FUNCTION_BLOCK PusherControl (* Basic Function Block Type *)
  (* Standard: 61499-2 *)
  (* Version 0.0, 1/14/2024, midxav, Template *)
  PACKAGE Main;
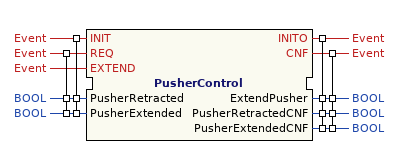
  EVENT_INPUT
    INIT WITH PusherRetracted, PusherExtended; (* Initialization Request *)
    REQ WITH PusherRetracted, PusherExtended; (* Normal Execution Request *)
    EXTEND;
  END_EVENT
  EVENT_OUTPUT
    INITO WITH ExtendPusher, PusherRetractedCNF, PusherExtendedCNF; (* Initialization Confirm *)
    CNF WITH ExtendPusher, PusherRetractedCNF, PusherExtendedCNF; (* Execution Confirmation *)
  END_EVENT
  VAR_INPUT
    PusherRetracted : BOOL;
    PusherExtended : BOOL;
  END_VAR
  VAR_OUTPUT
    ExtendPusher : BOOL;
    PusherRetractedCNF : BOOL;
    PusherExtendedCNF : BOOL;
  END_VAR
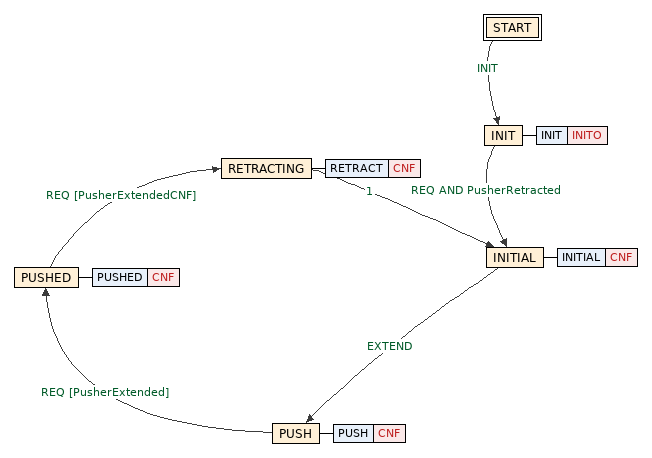
  EC_STATES
    START; (* Initial State *)
    INIT : INIT -> INITO; (* Initialization *)
    INITIAL : INITIAL -> CNF;
    PUSH : PUSH -> CNF;
    PUSHED : PUSHED -> CNF;
    RETRACTING : RETRACT -> CNF;
  END_STATES
  EC_TRANSITIONS
    START TO INIT := INIT;
    INIT TO INITIAL := REQ AND PusherRetracted;
    PUSH TO PUSHED := REQ [PusherExtended];
    INITIAL TO PUSH := EXTEND;
    PUSHED TO RETRACTING := REQ [PusherExtendedCNF];
    RETRACTING TO INITIAL := 1;
  END_TRANSITIONS
  ALGORITHM INIT IN ST: (* Initialization algorithm *)
ExtendPusher:= FALSE;
PusherExtendedCNF := FALSE;
PusherRetractedCNF := FALSE;
  END_ALGORITHM
  ALGORITHM PUSH IN ST:
ExtendPusher:=TRUE;
PusherRetractedCNF := FALSE;
  END_ALGORITHM
  ALGORITHM PUSHED IN ST:
ExtendPusher:=FALSE;
PusherExtendedCNF := TRUE;
  END_ALGORITHM
  ALGORITHM RETRACT IN ST:
;
PusherExtendedCNF := FALSE;
  END_ALGORITHM
  ALGORITHM INITIAL IN ST:
;
PusherRetractedCNF := TRUE;
PusherExtendedCNF := FALSE;
  END_ALGORITHM
END_FUNCTION_BLOCK
